{attribute 'qualified_only'}
{attribute 'strict'}
{attribute 'to_string'}
TYPE E_PMLUnitMode :
(
    Invalid			:= 0,	
    Production		:= 1,	//自動生産モード
    Maintenance		:= 2,	//保守・試運転モード
    Manual			:= 3	//手動JOG/単動モード
);
END_TYPE

(* stored: Version 1.1.0.1
   DUT E_PMLUnitMode: Id {27790a96-e13e-40b6-8c04-b0c688bde0df} *)
